Staubli VAL3: clkValve9.pgx

program clkValve9()
begin
  call toggleValve(9)
end
